Staubli VAL3: stop.pgx

public program stop()
begin
  SYS:doMouldFree[moduleIndex]=false
  SYS:doRobotOff[moduleIndex]=false
  SYS:doStartMachine[moduleIndex]=false
  bRobotOff=false
end
